% RSLogix 500 project P6.RSS, saved by version 12.00.00.00 %
PROJECT "UNTITLED"    % processor: Bul.1763 MicroLogix 1100 Series B %

PROGRAM FILES
  LAD 2   3 rungs
  LAD 3 "IO"  3 rungs
  LAD 4 "CTRL"  10 rungs

DATA FILES
  O0 OUTPUT  4 elements
  I1 INPUT  6 elements
  S2 STATUS  66 elements
  B3 BINARY  1 elements
  T4 TIMER  1 elements
  C5 COUNTER  3 elements
  R6 CONTROL  1 elements
  N7 INTEGER  4 elements
  F8 FLOAT  1 elements

LADDER 2
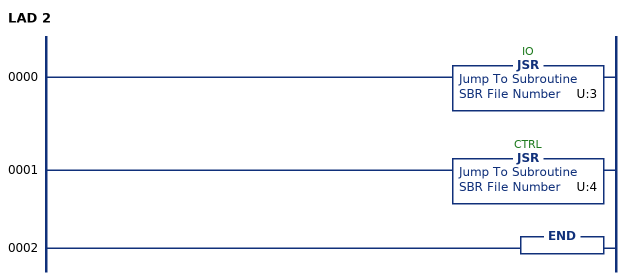
% Rung: 0 %
SOR JSR U:3 EOR
%   U:3  "IO" %
% Rung: 1 %
SOR JSR U:4 EOR
%   U:4  "CTRL" %
% Rung: 2 %
SOR END EOR

LADDER 3 "IO"
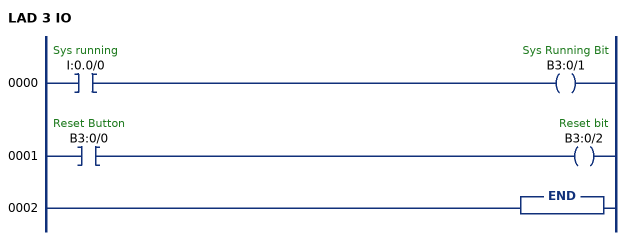
% Rung: 0 %
SOR XIC I:0.0/0 OTE B3:0/1 EOR
%   I:0.0/0  "Sys running" %
%   B3:0/1  "Sys Running Bit" %
% Rung: 1 %
SOR XIC B3:0/0 OTE B3:0/2 EOR
%   B3:0/0  "Reset Button" %
%   B3:0/2  "Reset bit" %
% Rung: 2 %
SOR END EOR

LADDER 4 "CTRL"
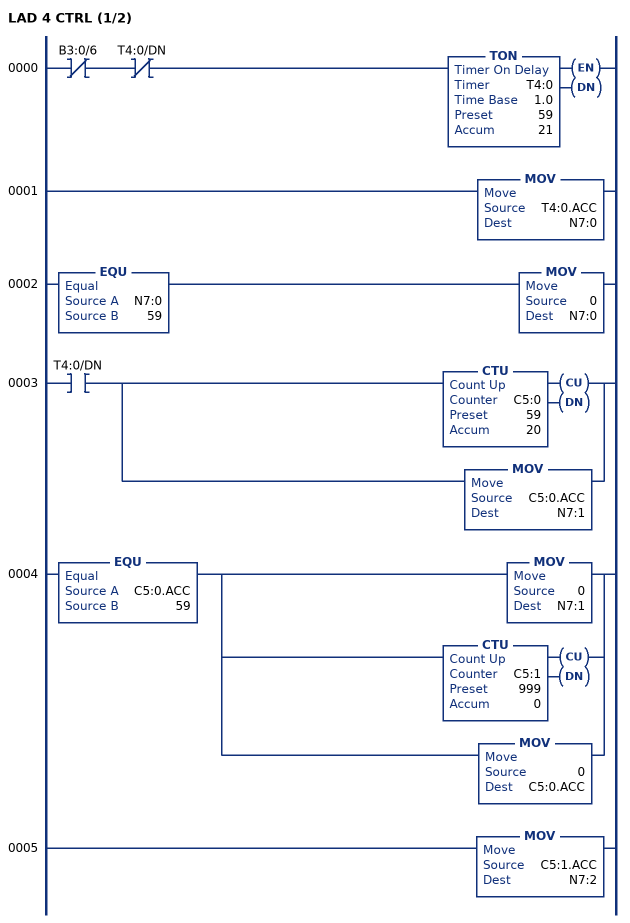
% Rung: 0 %
SOR XIO B3:0/6 XIO T4:0/DN TON T4:0 1.0 59 21 EOR
% Rung: 1 %
SOR MOV T4:0.ACC N7:0 EOR
% Rung: 2 %
SOR EQU N7:0 59 MOV 0 N7:0 EOR
% Rung: 3 %
SOR XIC T4:0/DN BST CTU C5:0 59 20 NXB MOV C5:0.ACC N7:1 BND EOR
% Rung: 4 %
SOR EQU C5:0.ACC 59 BST MOV 0 N7:1 NXB CTU C5:1 999 0 NXB MOV 0 C5:0.ACC BND EOR
% Rung: 5 %
SOR MOV C5:1.ACC N7:2 EOR

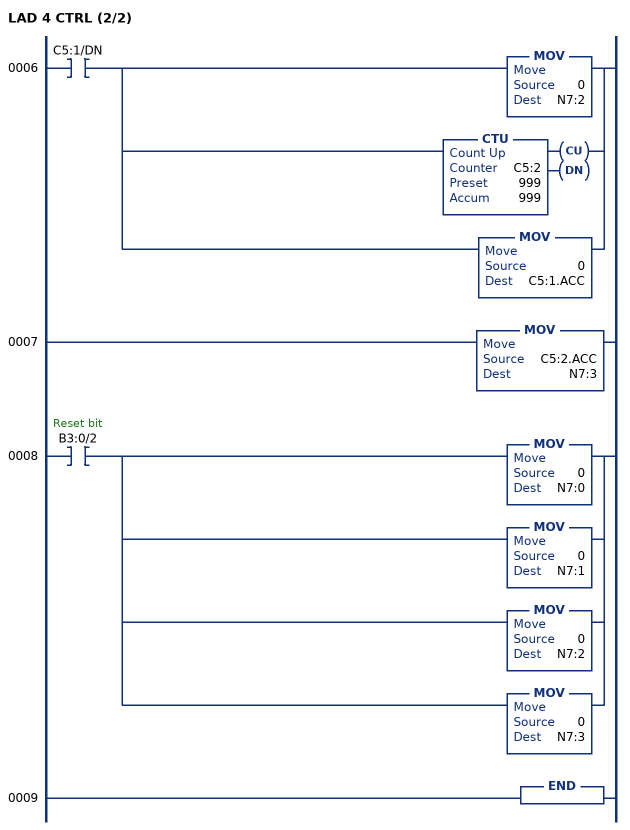
% Rung: 6 %
SOR XIC C5:1/DN BST MOV 0 N7:2 NXB CTU C5:2 999 999 NXB MOV 0 C5:1.ACC BND EOR
% Rung: 7 %
SOR MOV C5:2.ACC N7:3 EOR
% Rung: 8 %
SOR XIC B3:0/2 BST MOV 0 N7:0 NXB MOV 0 N7:1 NXB MOV 0 N7:2 NXB MOV 0 N7:3 BND EOR
%   B3:0/2  "Reset bit" %
% Rung: 9 %
SOR END EOR

OTHER DOCUMENTED ADDRESSES
  U2:0  "IO"
  U3:3  U3
  U3:4  U4

DATA TABLE (non-zero values as saved)
DATA T4
% .PRE .ACC %
% T4:0 % 59 21
DATA C5
% .PRE .ACC %
% C5:0 % 59 20
% C5:1 % 999 0
% C5:2 % 999 999
DATA N7
% N7:0 % 21 20 0 999
